// TIA Portal V18 export
DATA_BLOCK "L1_bkg"   // DB5
{ S7_Optimized_Access := 'TRUE' }
VERSION : 0.1
// stored: AutoNumber true, DBAccessibleFromOPCUA true, DBAccessibleFromWebserver true, IsOnlyStoredInLoadMemory false, IsRetainMemResEnabled false, IsWriteProtectedInAS false, MemoryReserve 100
   VAR RETAIN
      plcpc : "LGasp_type_Bck_visualizzazioni";
      pcplc : "LGasp_type_Bck_comandi";
   END_VAR
BEGIN
   // plcpc.visbool00[8] : Abilitazione operazioni compilazione
   // plcpc.visbool00[15] : richiesta esecuzione allargatura per semiauto
   // pcplc.cmdbool01[15] : risposta esecuzione allargatura per semiauto
   pcplc.cmdlreal[1] := 0.8;
   pcplc.cmdlreal[3] := 1.0;   // Correttore lunghezze mm
END_DATA_BLOCK
